Fanuc KAREL source: kt00295.KL

PROGRAM KT00295
%NOLOCKGROUP
VAR
I1:INTEGER
Y2 : ARRAY[2] OF BYTE
OUT:BOOLEAN
BEGIN
I1=2
Y2[1]=3
OUT=(I1<>Y2[1])
END KT00295
